TYPE TestStruct :
STRUCT
    {attribute 'pytmc' := '
        pv: Number
        io: i
     '}
    Number : LREAL;
    {attribute 'pytmc' := '
        pv: OK
        io: i
     '}
    Bin : BOOL;
END_STRUCT
END_TYPE

(* stored: Version 1.1.0.1, ProductVersion 3.1.4022.18
   DUT TestStruct: Id {c3e3d060-6cc0-4e43-adea-d4021a56a8cc} *)
